(* Logix 5000 project; controller STAT 1756-L72 rev 20.12; software revision 20.04; part 22 of 34 *)
(* tags used below, declared in another part *)
   DateTime : DINT[7];   // DINT array tag for retrieve wallclock time through GSV created during conversion
   I1 : INT[32];
   I10 : INT[2];
   I19 : INT[2];
   I2 : INT[2];
   I20_000 : ALIAS FOR I20[0];
   I20_001 : ALIAS FOR I20[1];
   I20_002 : ALIAS FOR I20[2];
   I20_003 : ALIAS FOR I20[3];
   I20_004 : ALIAS FOR I20[4];
   I20_005 : ALIAS FOR I20[5];
   I20_006 : ALIAS FOR I20[6];
   I20_007 : ALIAS FOR I20[7];
   I21_000 : ALIAS FOR I21[0];
   I21_001 : ALIAS FOR I21[1];
   I21_002 : ALIAS FOR I21[2];
   I21_003 : ALIAS FOR I21[3];
   I21_004 : ALIAS FOR I21[4];
   I21_005 : ALIAS FOR I21[5];
   I21_006 : ALIAS FOR I21[6];
   I21_007 : ALIAS FOR I21[7];
   I22_000 : ALIAS FOR I22[0];
   I22_001 : ALIAS FOR I22[1];
   I22_002 : ALIAS FOR I22[2];
   I22_003 : ALIAS FOR I22[3];
   I22_004 : ALIAS FOR I22[4];
   I22_005 : ALIAS FOR I22[5];
   I22_006 : ALIAS FOR I22[6];
   I22_007 : ALIAS FOR I22[7];
   I23_000 : ALIAS FOR I23[0];
   I23_001 : DINT;
   I23_002 : ALIAS FOR I23[2];
   I23_003 : ALIAS FOR I23[3];
   I23_004 : ALIAS FOR I23[4];
   I23_005 : ALIAS FOR I23[5];
   I23_006 : ALIAS FOR I23[6];
   I23_007 : DINT;
   I24_000 : ALIAS FOR I24[0];
   I24_001 : ALIAS FOR I24[1];
   I24_002 : ALIAS FOR I24[2];
   I24_003 : ALIAS FOR I24[3];
   I24_004 : ALIAS FOR I24[4];
   I24_005 : ALIAS FOR I24[5];
   I24_006 : ALIAS FOR I24[6];
   I24_007 : ALIAS FOR I24[7];
   I25_000 : ALIAS FOR I25[0];
   I25_001 : ALIAS FOR I25[1];
   I25_002 : ALIAS FOR I25[2];
   I25_003 : ALIAS FOR I25[3];
   I25_004 : ALIAS FOR I25[4];
   I25_005 : ALIAS FOR I25[5];
   I25_006 : ALIAS FOR I25[6];
   I25_007 : ALIAS FOR I25[7];
   I26_000 : ALIAS FOR I26[0];
   I26_001 : ALIAS FOR I26[1];
   I26_002 : ALIAS FOR I26[2];
   I26_003 : ALIAS FOR I26[3];
   I26_004 : ALIAS FOR I26[4];
   I26_005 : ALIAS FOR I26[5];
   I26_006 : ALIAS FOR I26[6];
   I26_007 : ALIAS FOR I26[7];
   I28_000 : ALIAS FOR I28[0];
   I28_001 : ALIAS FOR I28[1];
   I28_002 : ALIAS FOR I28[2];
   I28_003 : ALIAS FOR I28[3];
   I28_004 : ALIAS FOR I28[4];
   I28_005 : ALIAS FOR I28[5];
   I28_006 : ALIAS FOR I28[6];
   I28_007 : ALIAS FOR I28[7];
   I3 : INT[2];
   I4 : INT[2];
   I5 : INT[2];
   I6 : INT[2];
   I7 : INT[2];
   I8 : INT[2];
   I9 : INT[2];
   inb : DINT;
   N19 : DINT[80];
   N20 : DINT[80];
   N21 : DINT[80];
   N23 : DINT[80];
   N24 : DINT[80];
   N7 : DINT[255];
   O1 : INT[32];
   O12 : INT[2];
   O13 : INT[2];
   O14 : INT[2];
   O15 : INT[2];
   O16 : INT[2];
   O17 : INT[2];
   O18 : INT[2];
   O27_000 : ALIAS FOR O27[0];
   O27_001 : ALIAS FOR O27[1];
   O27_002 : ALIAS FOR O27[2];
   O27_003 : ALIAS FOR O27[3];
   Seconde : BOOL;
(* ibt, continued *)

ROUTINE ibtmain   (* ladder *)
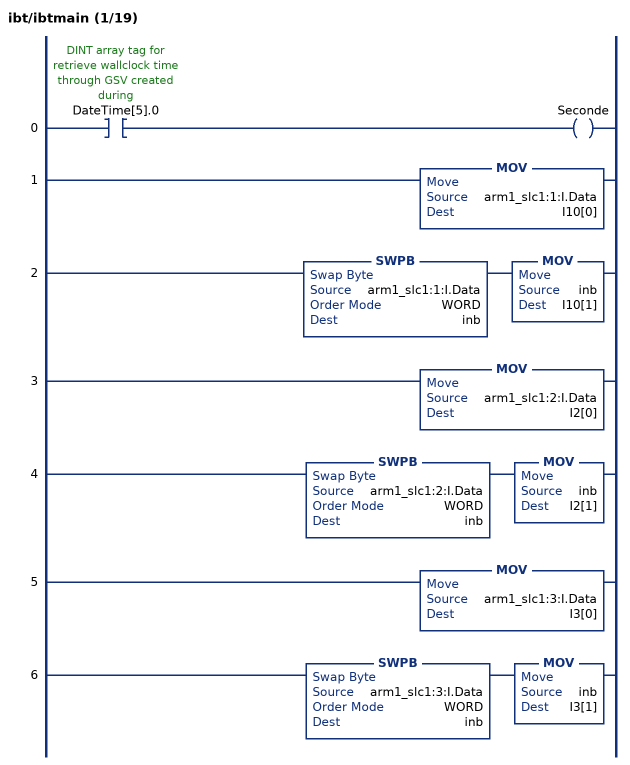
   0: XIC(DateTime[5].0)OTE(Seconde);
   1: MOV(arm1_slc1:1:I.Data,I10[0]);
   2: SWPB(arm1_slc1:1:I.Data,WORD,inb)MOV(inb,I10[1]);
   3: MOV(arm1_slc1:2:I.Data,I2[0]);
   4: SWPB(arm1_slc1:2:I.Data,WORD,inb)MOV(inb,I2[1]);
   5: MOV(arm1_slc1:3:I.Data,I3[0]);
   6: SWPB(arm1_slc1:3:I.Data,WORD,inb)MOV(inb,I3[1]);
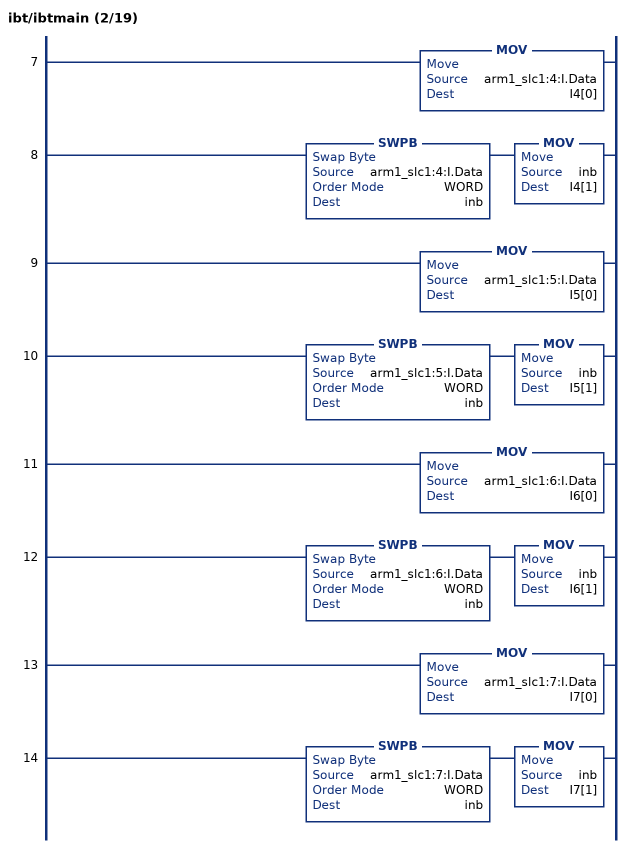
   7: MOV(arm1_slc1:4:I.Data,I4[0]);
   8: SWPB(arm1_slc1:4:I.Data,WORD,inb)MOV(inb,I4[1]);
   9: MOV(arm1_slc1:5:I.Data,I5[0]);
   10: SWPB(arm1_slc1:5:I.Data,WORD,inb)MOV(inb,I5[1]);
   11: MOV(arm1_slc1:6:I.Data,I6[0]);
   12: SWPB(arm1_slc1:6:I.Data,WORD,inb)MOV(inb,I6[1]);
   13: MOV(arm1_slc1:7:I.Data,I7[0]);
   14: SWPB(arm1_slc1:7:I.Data,WORD,inb)MOV(inb,I7[1]);
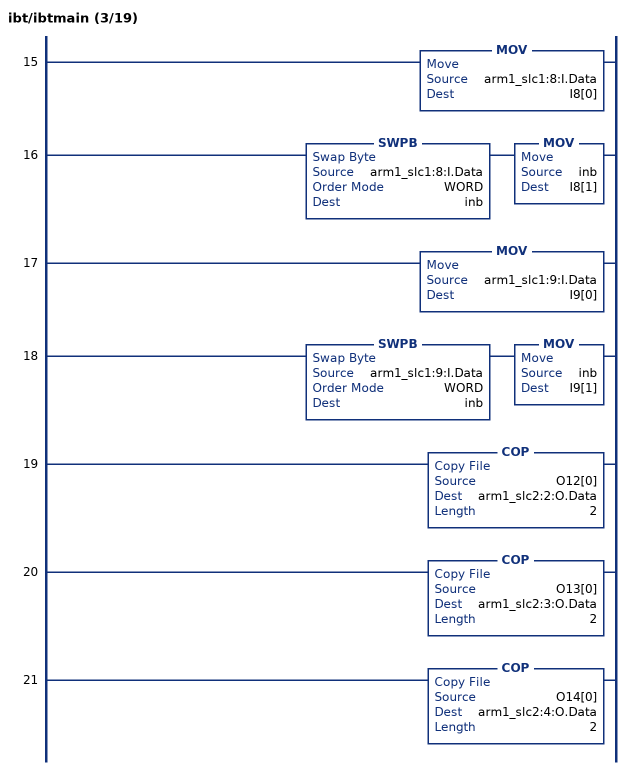
   15: MOV(arm1_slc1:8:I.Data,I8[0]);
   16: SWPB(arm1_slc1:8:I.Data,WORD,inb)MOV(inb,I8[1]);
   17: MOV(arm1_slc1:9:I.Data,I9[0]);
   18: SWPB(arm1_slc1:9:I.Data,WORD,inb)MOV(inb,I9[1]);
   19: COP(O12[0],arm1_slc2:2:O.Data,2);
   20: COP(O13[0],arm1_slc2:3:O.Data,2);
   21: COP(O14[0],arm1_slc2:4:O.Data,2);
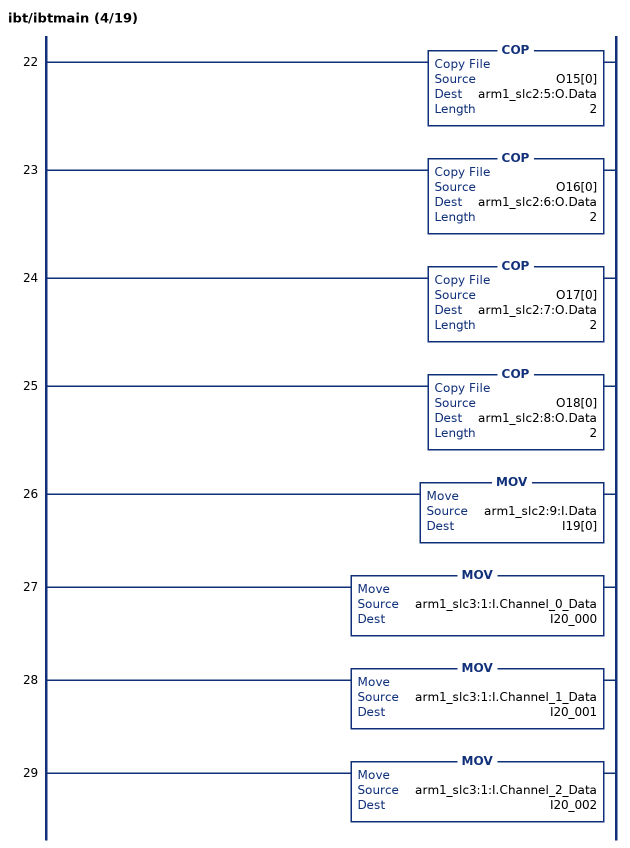
   22: COP(O15[0],arm1_slc2:5:O.Data,2);
   23: COP(O16[0],arm1_slc2:6:O.Data,2);
   24: COP(O17[0],arm1_slc2:7:O.Data,2);
   25: COP(O18[0],arm1_slc2:8:O.Data,2);
   26: MOV(arm1_slc2:9:I.Data,I19[0]);
   27: MOV(arm1_slc3:1:I.Channel_0_Data,I20_000);
   28: MOV(arm1_slc3:1:I.Channel_1_Data,I20_001);
   29: MOV(arm1_slc3:1:I.Channel_2_Data,I20_002);
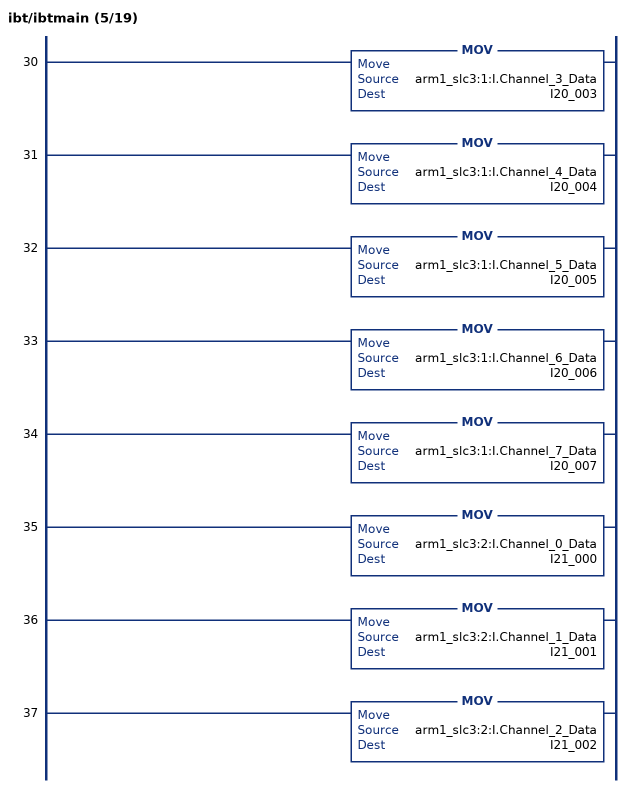
   30: MOV(arm1_slc3:1:I.Channel_3_Data,I20_003);
   31: MOV(arm1_slc3:1:I.Channel_4_Data,I20_004);
   32: MOV(arm1_slc3:1:I.Channel_5_Data,I20_005);
   33: MOV(arm1_slc3:1:I.Channel_6_Data,I20_006);
   34: MOV(arm1_slc3:1:I.Channel_7_Data,I20_007);
   35: MOV(arm1_slc3:2:I.Channel_0_Data,I21_000);
   36: MOV(arm1_slc3:2:I.Channel_1_Data,I21_001);
   37: MOV(arm1_slc3:2:I.Channel_2_Data,I21_002);
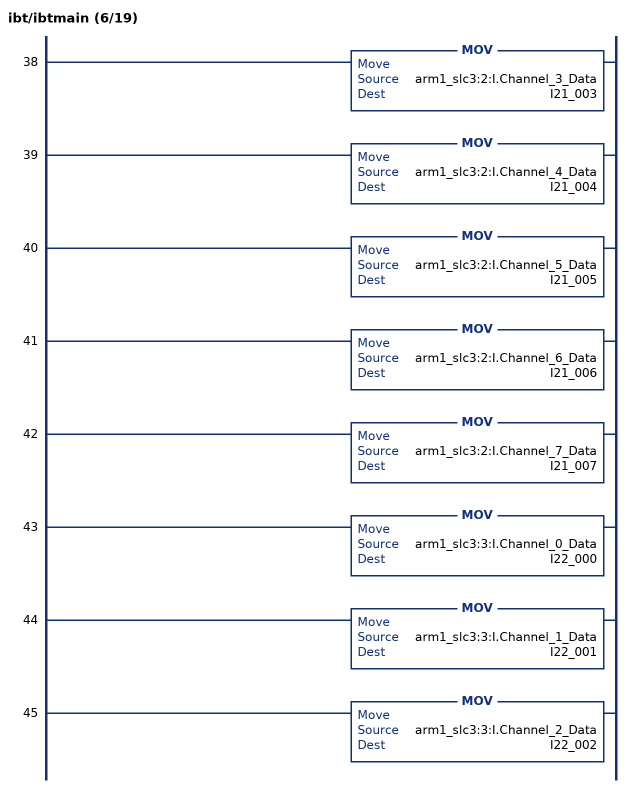
   38: MOV(arm1_slc3:2:I.Channel_3_Data,I21_003);
   39: MOV(arm1_slc3:2:I.Channel_4_Data,I21_004);
   40: MOV(arm1_slc3:2:I.Channel_5_Data,I21_005);
   41: MOV(arm1_slc3:2:I.Channel_6_Data,I21_006);
   42: MOV(arm1_slc3:2:I.Channel_7_Data,I21_007);
   43: MOV(arm1_slc3:3:I.Channel_0_Data,I22_000);
   44: MOV(arm1_slc3:3:I.Channel_1_Data,I22_001);
   45: MOV(arm1_slc3:3:I.Channel_2_Data,I22_002);
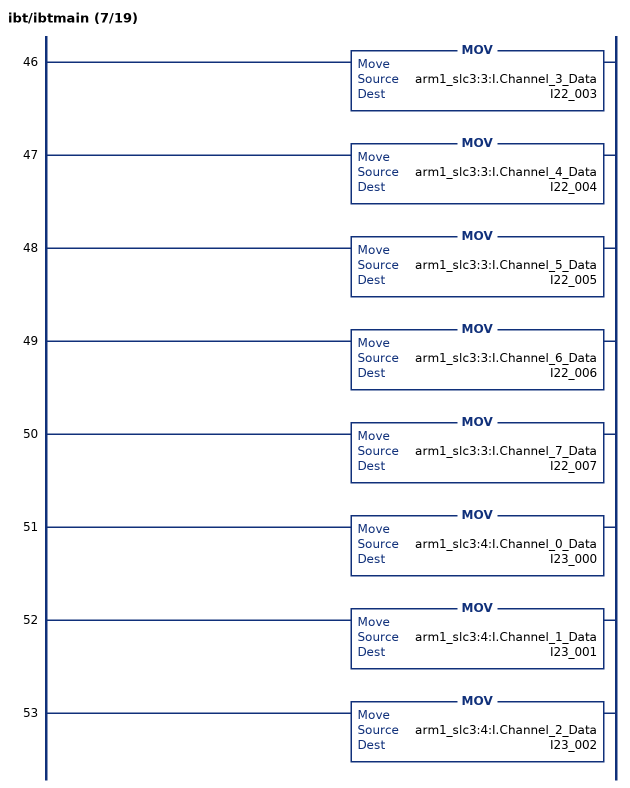
   46: MOV(arm1_slc3:3:I.Channel_3_Data,I22_003);
   47: MOV(arm1_slc3:3:I.Channel_4_Data,I22_004);
   48: MOV(arm1_slc3:3:I.Channel_5_Data,I22_005);
   49: MOV(arm1_slc3:3:I.Channel_6_Data,I22_006);
   50: MOV(arm1_slc3:3:I.Channel_7_Data,I22_007);
   51: MOV(arm1_slc3:4:I.Channel_0_Data,I23_000);
   52: MOV(arm1_slc3:4:I.Channel_1_Data,I23_001);
   53: MOV(arm1_slc3:4:I.Channel_2_Data,I23_002);
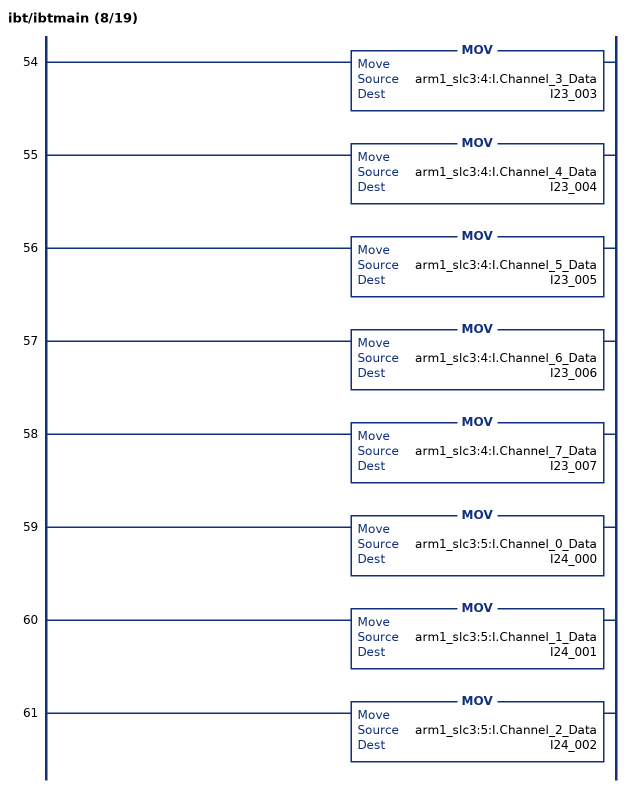
   54: MOV(arm1_slc3:4:I.Channel_3_Data,I23_003);
   55: MOV(arm1_slc3:4:I.Channel_4_Data,I23_004);
   56: MOV(arm1_slc3:4:I.Channel_5_Data,I23_005);
   57: MOV(arm1_slc3:4:I.Channel_6_Data,I23_006);
   58: MOV(arm1_slc3:4:I.Channel_7_Data,I23_007);
   59: MOV(arm1_slc3:5:I.Channel_0_Data,I24_000);
   60: MOV(arm1_slc3:5:I.Channel_1_Data,I24_001);
   61: MOV(arm1_slc3:5:I.Channel_2_Data,I24_002);
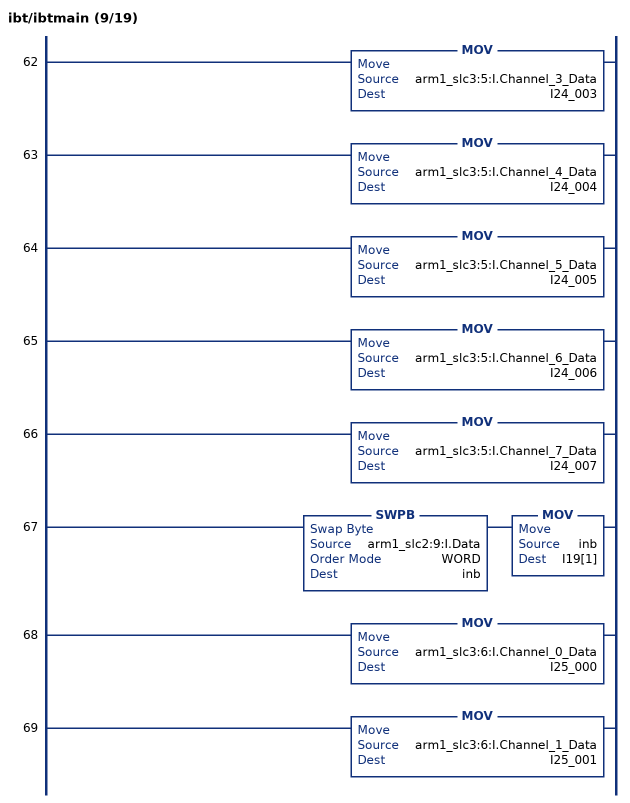
   62: MOV(arm1_slc3:5:I.Channel_3_Data,I24_003);
   63: MOV(arm1_slc3:5:I.Channel_4_Data,I24_004);
   64: MOV(arm1_slc3:5:I.Channel_5_Data,I24_005);
   65: MOV(arm1_slc3:5:I.Channel_6_Data,I24_006);
   66: MOV(arm1_slc3:5:I.Channel_7_Data,I24_007);
   67: SWPB(arm1_slc2:9:I.Data,WORD,inb)MOV(inb,I19[1]);
   68: MOV(arm1_slc3:6:I.Channel_0_Data,I25_000);
   69: MOV(arm1_slc3:6:I.Channel_1_Data,I25_001);
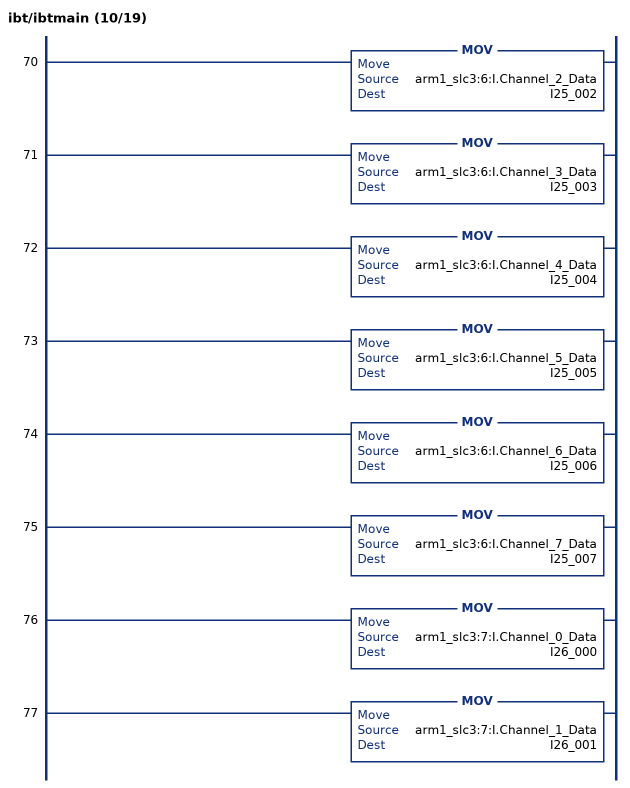
   70: MOV(arm1_slc3:6:I.Channel_2_Data,I25_002);
   71: MOV(arm1_slc3:6:I.Channel_3_Data,I25_003);
   72: MOV(arm1_slc3:6:I.Channel_4_Data,I25_004);
   73: MOV(arm1_slc3:6:I.Channel_5_Data,I25_005);
   74: MOV(arm1_slc3:6:I.Channel_6_Data,I25_006);
   75: MOV(arm1_slc3:6:I.Channel_7_Data,I25_007);
   76: MOV(arm1_slc3:7:I.Channel_0_Data,I26_000);
   77: MOV(arm1_slc3:7:I.Channel_1_Data,I26_001);
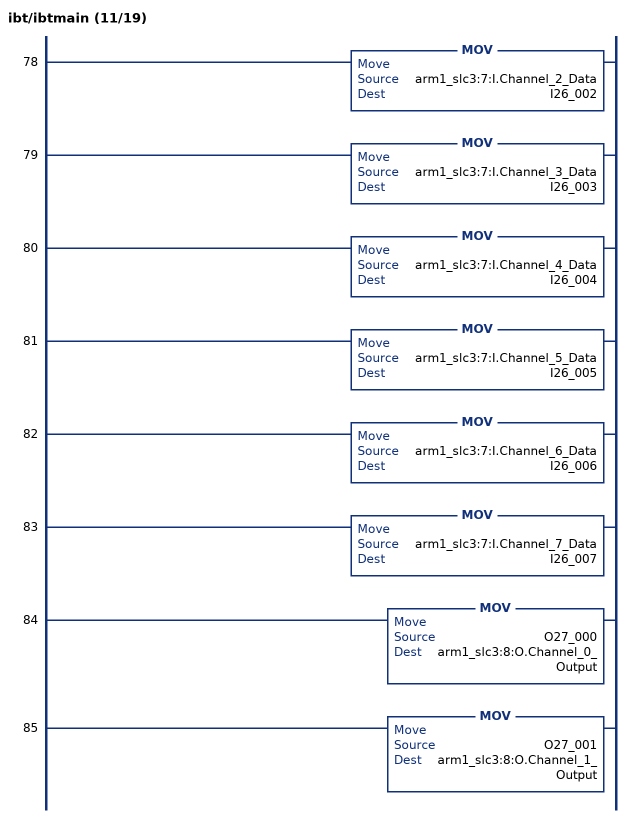
   78: MOV(arm1_slc3:7:I.Channel_2_Data,I26_002);
   79: MOV(arm1_slc3:7:I.Channel_3_Data,I26_003);
   80: MOV(arm1_slc3:7:I.Channel_4_Data,I26_004);
   81: MOV(arm1_slc3:7:I.Channel_5_Data,I26_005);
   82: MOV(arm1_slc3:7:I.Channel_6_Data,I26_006);
   83: MOV(arm1_slc3:7:I.Channel_7_Data,I26_007);
   84: MOV(O27_000,arm1_slc3:8:O.Channel_0_Output);
   85: MOV(O27_001,arm1_slc3:8:O.Channel_1_Output);
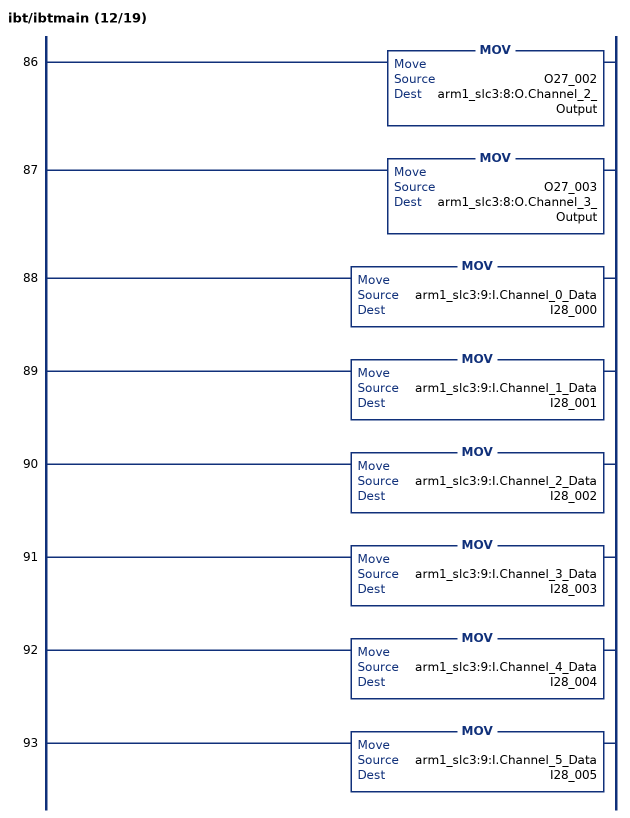
   86: MOV(O27_002,arm1_slc3:8:O.Channel_2_Output);
   87: MOV(O27_003,arm1_slc3:8:O.Channel_3_Output);
   88: MOV(arm1_slc3:9:I.Channel_0_Data,I28_000);
   89: MOV(arm1_slc3:9:I.Channel_1_Data,I28_001);
   90: MOV(arm1_slc3:9:I.Channel_2_Data,I28_002);
   91: MOV(arm1_slc3:9:I.Channel_3_Data,I28_003);
   92: MOV(arm1_slc3:9:I.Channel_4_Data,I28_004);
   93: MOV(arm1_slc3:9:I.Channel_5_Data,I28_005);
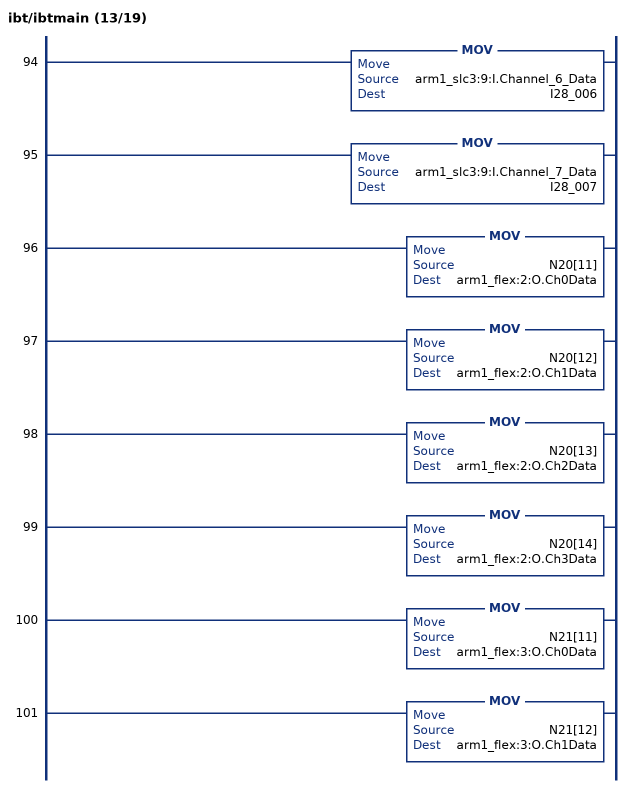
   94: MOV(arm1_slc3:9:I.Channel_6_Data,I28_006);
   95: MOV(arm1_slc3:9:I.Channel_7_Data,I28_007);
   96: MOV(N20[11],arm1_flex:2:O.Ch0Data);
   97: MOV(N20[12],arm1_flex:2:O.Ch1Data);
   98: MOV(N20[13],arm1_flex:2:O.Ch2Data);
   99: MOV(N20[14],arm1_flex:2:O.Ch3Data);
   100: MOV(N21[11],arm1_flex:3:O.Ch0Data);
   101: MOV(N21[12],arm1_flex:3:O.Ch1Data);
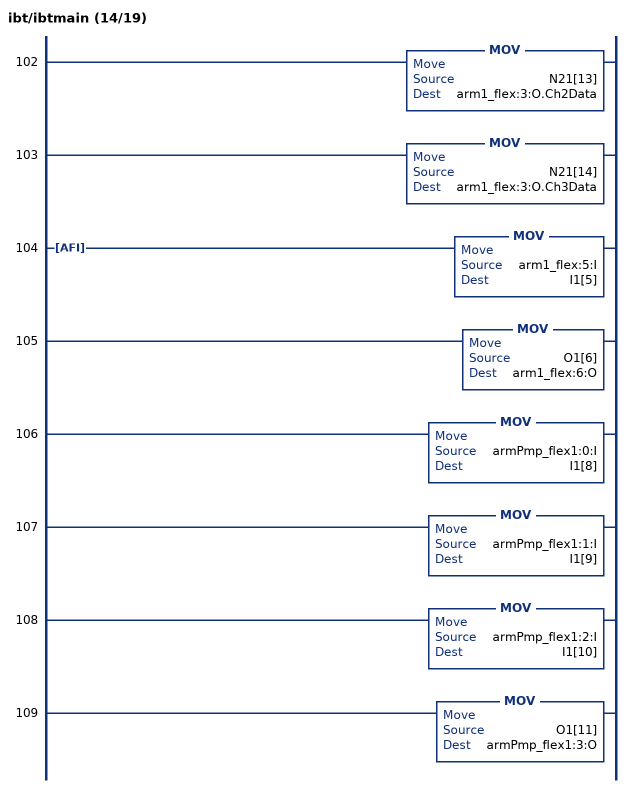
   102: MOV(N21[13],arm1_flex:3:O.Ch2Data);
   103: MOV(N21[14],arm1_flex:3:O.Ch3Data);
   104: AFI()MOV(arm1_flex:5:I,I1[5]);
   105: MOV(O1[6],arm1_flex:6:O);
   106: MOV(armPmp_flex1:0:I,I1[8]);
   107: MOV(armPmp_flex1:1:I,I1[9]);
   108: MOV(armPmp_flex1:2:I,I1[10]);
   109: MOV(O1[11],armPmp_flex1:3:O);
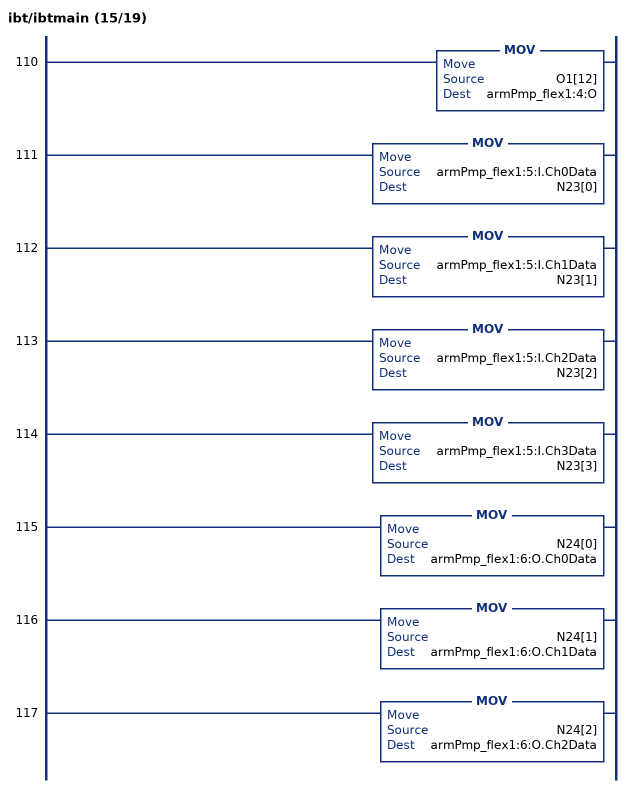
   110: MOV(O1[12],armPmp_flex1:4:O);
   111: MOV(armPmp_flex1:5:I.Ch0Data,N23[0]);
   112: MOV(armPmp_flex1:5:I.Ch1Data,N23[1]);
   113: MOV(armPmp_flex1:5:I.Ch2Data,N23[2]);
   114: MOV(armPmp_flex1:5:I.Ch3Data,N23[3]);
   115: MOV(N24[0],armPmp_flex1:6:O.Ch0Data);
   116: MOV(N24[1],armPmp_flex1:6:O.Ch1Data);
   117: MOV(N24[2],armPmp_flex1:6:O.Ch2Data);
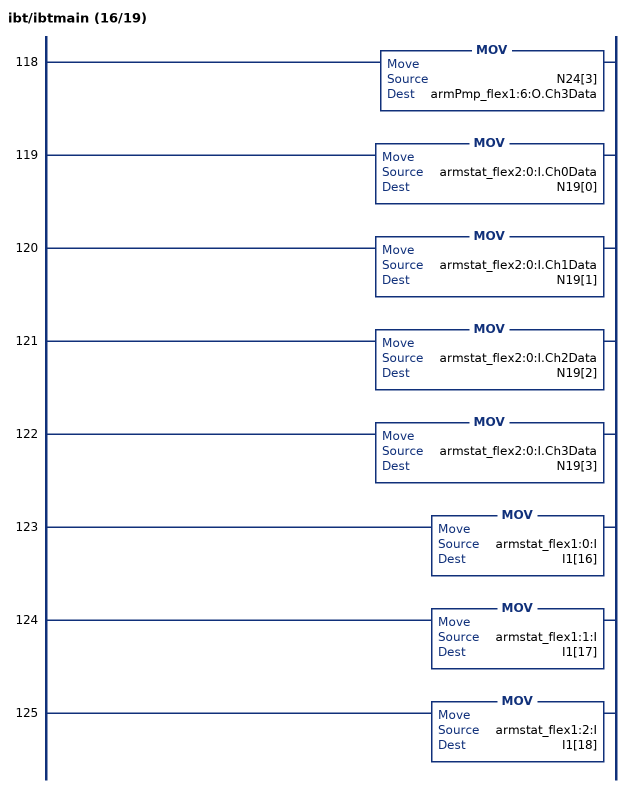
   118: MOV(N24[3],armPmp_flex1:6:O.Ch3Data);
   119: MOV(armstat_flex2:0:I.Ch0Data,N19[0]);
   120: MOV(armstat_flex2:0:I.Ch1Data,N19[1]);
   121: MOV(armstat_flex2:0:I.Ch2Data,N19[2]);
   122: MOV(armstat_flex2:0:I.Ch3Data,N19[3]);
   123: MOV(armstat_flex1:0:I,I1[16]);
   124: MOV(armstat_flex1:1:I,I1[17]);
   125: MOV(armstat_flex1:2:I,I1[18]);
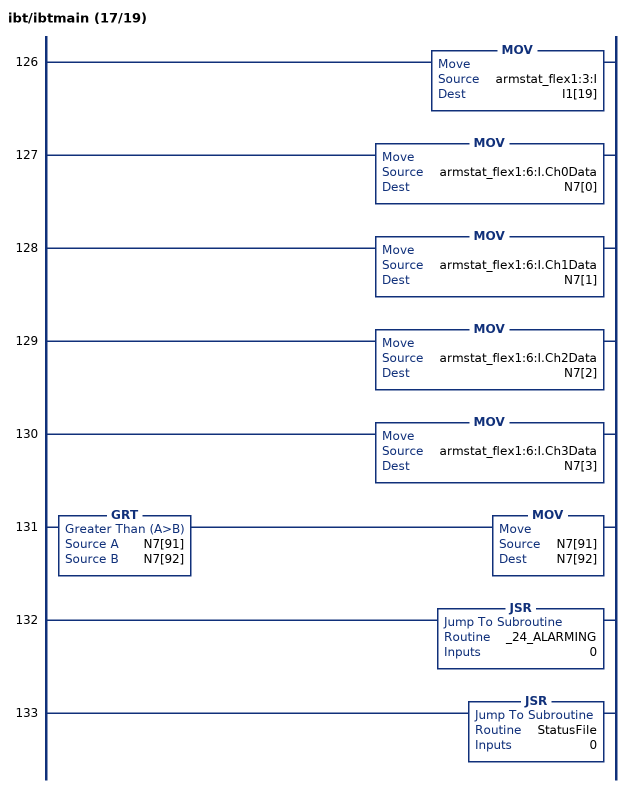
   126: MOV(armstat_flex1:3:I,I1[19]);
   127: MOV(armstat_flex1:6:I.Ch0Data,N7[0]);
   128: MOV(armstat_flex1:6:I.Ch1Data,N7[1]);
   129: MOV(armstat_flex1:6:I.Ch2Data,N7[2]);
   130: MOV(armstat_flex1:6:I.Ch3Data,N7[3]);
   131: GRT(N7[91],N7[92])MOV(N7[91],N7[92]);
   132: JSR(_24_ALARMING,0);
   133: JSR(StatusFile,0);
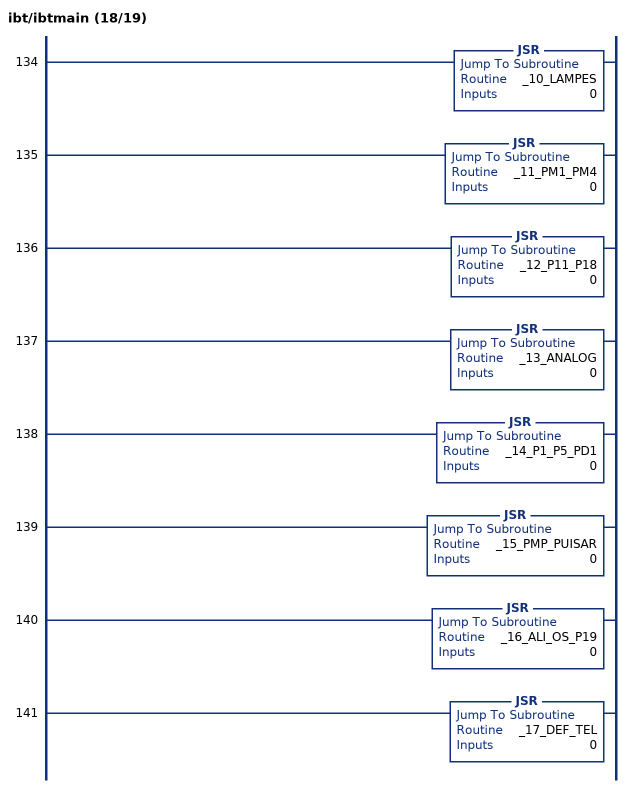
   134: JSR(_10_LAMPES,0);
   135: JSR(_11_PM1_PM4,0);
   136: JSR(_12_P11_P18,0);
   137: JSR(_13_ANALOG,0);
   138: JSR(_14_P1_P5_PD1,0);
   139: JSR(_15_PMP_PUISAR,0);
   140: JSR(_16_ALI_OS_P19,0);
   141: JSR(_17_DEF_TEL,0);
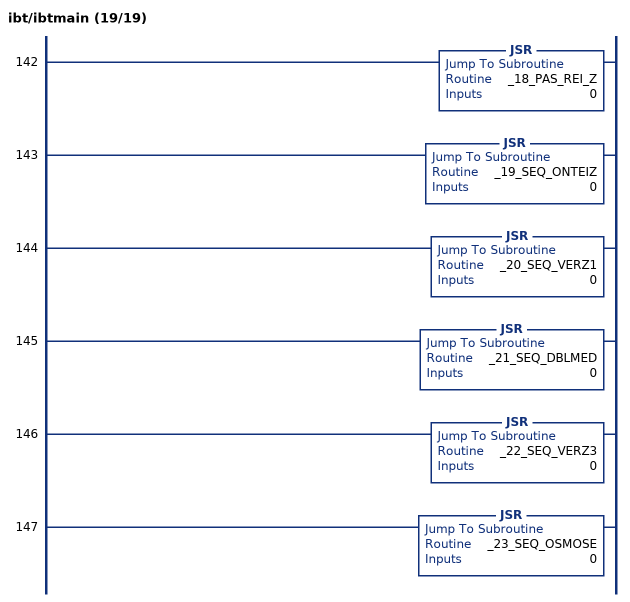
   142: JSR(_18_PAS_REI_Z,0);
   143: JSR(_19_SEQ_ONTEIZ,0);
   144: JSR(_20_SEQ_VERZ1,0);
   145: JSR(_21_SEQ_DBLMED,0);
   146: JSR(_22_SEQ_VERZ3,0);
   147: JSR(_23_SEQ_OSMOSE,0);
END_ROUTINE
